// Encode a 32-BIT value with ZigZag encoding.
FUNCTION F_EncodeZigZag32 : UDINT
VAR_INPUT
    nValue : DINT;
END_VAR

F_EncodeZigZag32 := TO_UDINT(SHL(nValue, 1)) XOR TO_UDINT(SHR(nValue, 31));

END_FUNCTION

(* stored: Version 1.1.0.1
   POU F_EncodeZigZag32: Id {6e2eb686-b576-46ba-842c-7a9c56e8b00c}, SpecialFunc None *)
